// Mitsubishi GX Works2 project: BTL_FX2N   PLC: FX2N/FX2NC

PROGRAM MAIN
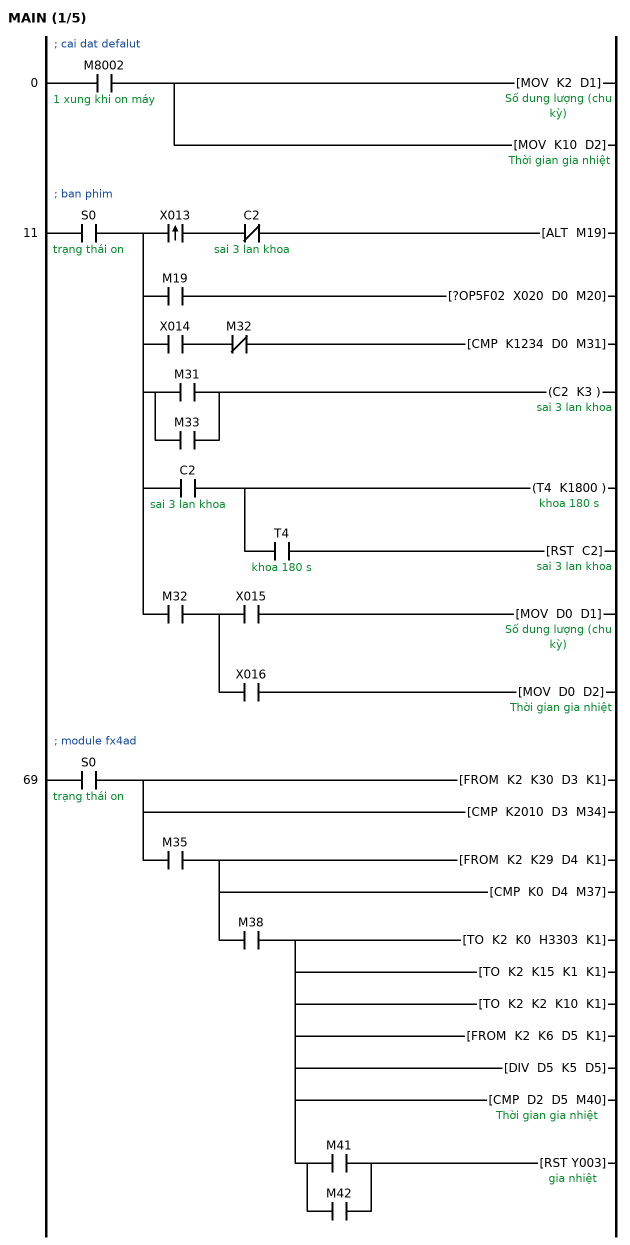
; cai dat defalut
0     LD      M8002  ; 1 xung khi on máy
      MOV     K2 D1  ; Số dung lượng (chu kỳ)
      MOV     K10 D2  ; Thời gian gia nhiệt
; ban phim
11    LD      S0  ; trạng thái on
      MPS
      ANDP    X013
      ANI     C2  ; sai 3 lan khoa
      ALT     M19
      MRD
      AND     M19
      ?OP5F02 X020 D0 M20
      MRD
      AND     X014
      ANI     M32
      CMP     K1234 D0 M31
      MRD
      LD      M31
      OR      M33
      ANB
      OUT     C2 K3  ; sai 3 lan khoa
      MRD
      AND     C2  ; sai 3 lan khoa
      OUT     T4 K1800  ; khoa 180 s
      AND     T4  ; khoa 180 s
      RST     C2  ; sai 3 lan khoa
      MPP
      AND     M32
      MPS
      AND     X015
      MOV     D0 D1
      MPP
      AND     X016
      MOV     D0 D2
; module fx4ad
69    LD      S0  ; trạng thái on
      FROM    K2 K30 D3 K1
        [note] lay BF30 nhan dang
      CMP     K2010 D3 M34
        [note] check fx4ad
      AND     M35
      FROM    K2 K29 D4 K1
        [note] lay du lieu loi BF29
      CMP     K0 D4 M37
        [note] khong co loi
      AND     M38
      TO      K2 K0 H3303 K1
        [note] khoi tao CH2 BF#0
      TO      K2 K15 K1 K1
        [note] toc do cao BF15 6ms
      TO      K2 K2 K10 K1
        [note] so luong lay mau CH2 la 10
      FROM    K2 K6 D5 K1
        [note] lay nhiet do trung binh vao D5
      DIV     D5 K5 D5
        [note] chia calib +-400 voi +-2000
      CMP     D2 D5 M40
      LD      M41
      OR      M42
      ANB
      RST     Y003  ; gia nhiệt
        [note] bang hoac cao hon thi tat
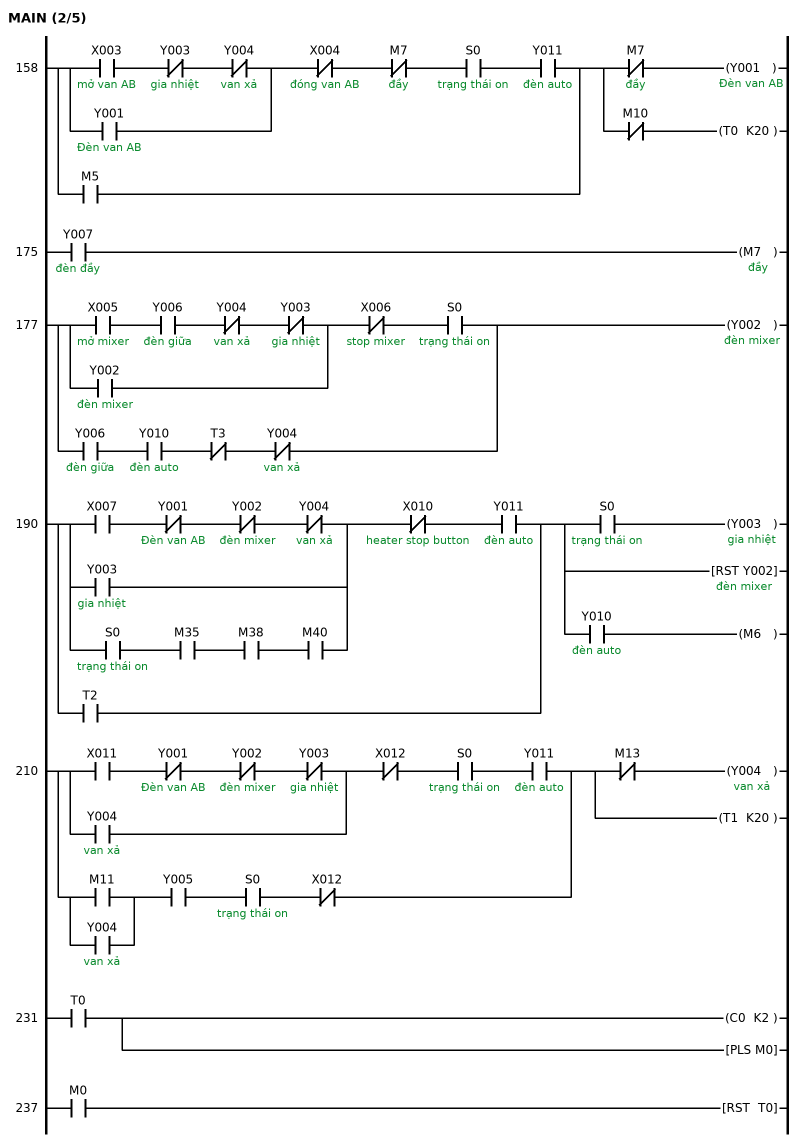
158   LD      X003  ; mở van AB
      ANI     Y003  ; gia nhiệt
      ANI     Y004  ; van xả
      OR      Y001  ; Đèn van AB
      ANI     X004  ; đóng van AB
      ANI     M7  ; đầy
      AND     S0  ; trạng thái on
      AND     Y011  ; đèn auto
      OR      M5
      MPS
      ANI     M7  ; đầy
      OUT     Y001  ; Đèn van AB
      MPP
      ANI     M10
      OUT     T0 K20
175   LD      Y007  ; đèn đầy
      OUT     M7  ; đầy
177   LD      X005  ; mở mixer
      AND     Y006  ; đèn giữa
      ANI     Y004  ; van xả
      ANI     Y003  ; gia nhiệt
      OR      Y002  ; đèn mixer
      ANI     X006  ; stop mixer
      AND     S0  ; trạng thái on
      LD      Y006  ; đèn giữa
      AND     Y010  ; đèn auto
      ANI     T3
      ANI     Y004  ; van xả
      ORB
      OUT     Y002  ; đèn mixer
190   LD      X007
      ANI     Y001  ; Đèn van AB
      ANI     Y002  ; đèn mixer
      ANI     Y004  ; van xả
      OR      Y003  ; gia nhiệt
      LD      S0  ; trạng thái on
      AND     M35
      AND     M38
      AND     M40
      ORB
      ANI     X010  ; heater stop button
      AND     Y011  ; đèn auto
      OR      T2
      MPS
      AND     S0  ; trạng thái on
      OUT     Y003  ; gia nhiệt
      MPP
      RST     Y002  ; đèn mixer
      AND     Y010  ; đèn auto
      OUT     M6
210   LD      X011
      ANI     Y001  ; Đèn van AB
      ANI     Y002  ; đèn mixer
      ANI     Y003  ; gia nhiệt
      OR      Y004  ; van xả
      ANI     X012
      AND     S0  ; trạng thái on
      AND     Y011  ; đèn auto
      LD      M11
      OR      Y004  ; van xả
      AND     Y005
      AND     S0  ; trạng thái on
      ANI     X012
      ORB
      MPS
      ANI     M13
      OUT     Y004  ; van xả
      MPP
      OUT     T1 K20
231   LD      T0
      OUT     C0 K2
      PLS     M0
237   LD      M0
      RST     T0
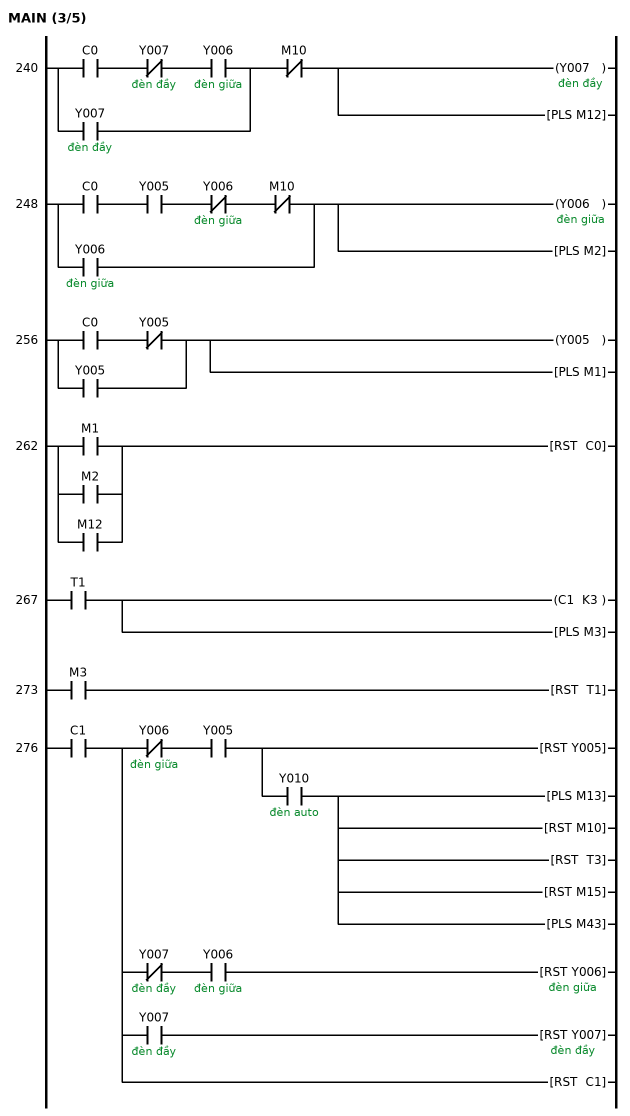
240   LD      C0
      ANI     Y007  ; đèn đầy
      AND     Y006  ; đèn giữa
      OR      Y007  ; đèn đầy
      ANI     M10
      OUT     Y007  ; đèn đầy
      PLS     M12
248   LD      C0
      AND     Y005
      ANI     Y006  ; đèn giữa
      ANI     M10
      OR      Y006  ; đèn giữa
      OUT     Y006  ; đèn giữa
      PLS     M2
256   LD      C0
      ANI     Y005
      OR      Y005
      OUT     Y005
      PLS     M1
262   LD      M1
      OR      M2
      OR      M12
      RST     C0
267   LD      T1
      OUT     C1 K3
      PLS     M3
273   LD      M3
      RST     T1
276   LD      C1
      MPS
      ANI     Y006  ; đèn giữa
      AND     Y005
      RST     Y005
      AND     Y010  ; đèn auto
      PLS     M13
      RST     M10
      RST     T3
      RST     M15
      PLS     M43
      MRD
      ANI     Y007  ; đèn đầy
      AND     Y006  ; đèn giữa
      RST     Y006  ; đèn giữa
      MRD
      AND     Y007  ; đèn đầy
      RST     Y007  ; đèn đầy
      MPP
      RST     C1
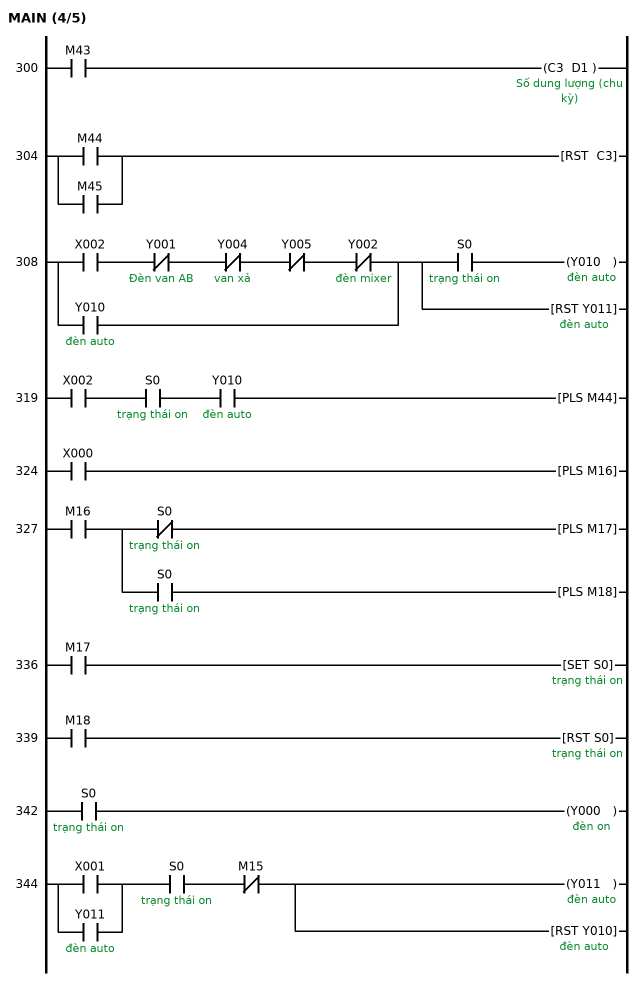
300   LD      M43
      OUT     C3 D1  ; Số dung lượng (chu kỳ)
304   LD      M44
      OR      M45
      RST     C3
308   LD      X002
      ANI     Y001  ; Đèn van AB
      ANI     Y004  ; van xả
      ANI     Y005
      ANI     Y002  ; đèn mixer
      OR      Y010  ; đèn auto
      MPS
      AND     S0  ; trạng thái on
      OUT     Y010  ; đèn auto
      MPP
      RST     Y011  ; đèn auto
319   LD      X002
      AND     S0  ; trạng thái on
      AND     Y010  ; đèn auto
      PLS     M44
324   LD      X000
      PLS     M16
327   LD      M16
      MPS
      ANI     S0  ; trạng thái on
      PLS     M17
      MPP
      AND     S0  ; trạng thái on
      PLS     M18
336   LD      M17
      SET     S0  ; trạng thái on
339   LD      M18
      RST     S0  ; trạng thái on
342   LD      S0  ; trạng thái on
      OUT     Y000  ; đèn on
344   LD      X001
      OR      Y011  ; đèn auto
      AND     S0  ; trạng thái on
      ANI     M15
      OUT     Y011  ; đèn auto
      RST     Y010  ; đèn auto
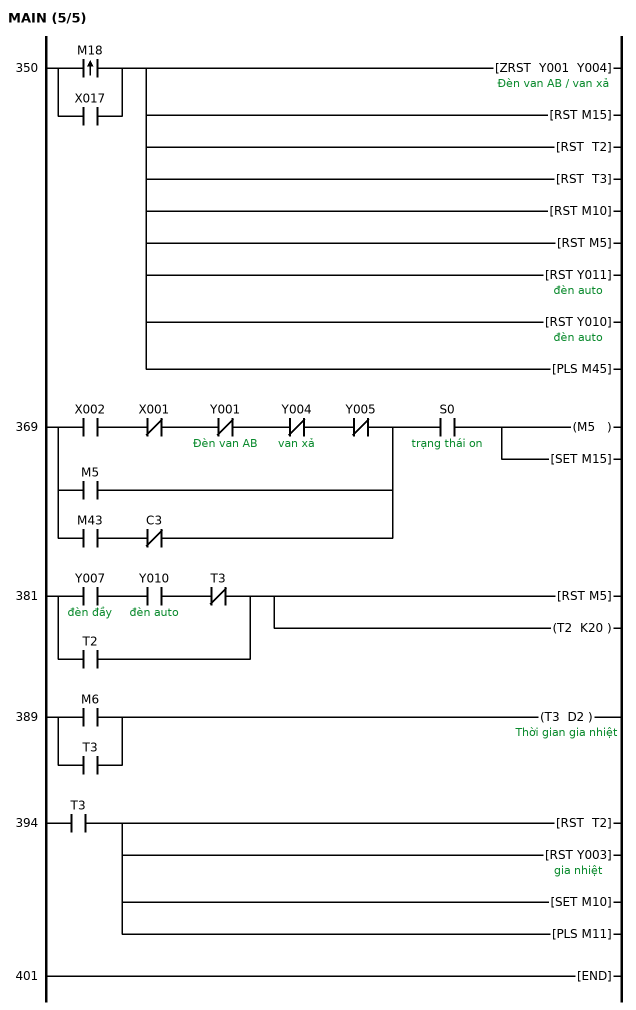
350   LDP     M18
      OR      X017
      ZRST    Y001 Y004
      RST     M15
      RST     T2
      RST     T3
      RST     M10
      RST     M5
      RST     Y011  ; đèn auto
      RST     Y010  ; đèn auto
      PLS     M45
369   LD      X002
      ANI     X001
      ANI     Y001  ; Đèn van AB
      ANI     Y004  ; van xả
      ANI     Y005
      OR      M5
      LD      M43
      ANI     C3
      ORB
      AND     S0  ; trạng thái on
      OUT     M5
      SET     M15
381   LD      Y007  ; đèn đầy
      AND     Y010  ; đèn auto
      ANI     T3
      OR      T2
      RST     M5
      OUT     T2 K20
389   LD      M6
      OR      T3
      OUT     T3 D2  ; Thời gian gia nhiệt
394   LD      T3
      RST     T2
      RST     Y003  ; gia nhiệt
      SET     M10
      PLS     M11
401   END
END_PROGRAM
